TYPE "udt_RollLubr_Valve_Pers"
VERSION : 0.1
// Block: udt_RollLubr_Valve_Pers
   STRUCT
      SystemOn : Bool;
      Enable_V : Array[1..ROLL_LUBR_MAXVALVE] of Bool;
      TimeOn : Time;
      TimeOff : Time;
   END_STRUCT;

END_TYPE
